// TIA Portal project "tamp" (V16)

(* hardware
DEVICE "S7-1200 station_1"  S7-1200 Station
   slot 0: "Rack_0"  S7-1200 Rack  Rack  V1.0
   slot 1: "PLC_1"  CPU 1212C AC/DC/Rly  6ES7 212-1BE40-0XB0  V4.0
*)

// ===== PLC "PLC_1"  CPU 1212C AC/DC/Rly =====

VAR_GLOBAL   // PLC tag table "Default tag table"
   "K1" AT %Q0.0 : Bool;
   "stop1" AT %I0.4 : Bool;
   "k2" AT %Q0.1 : Bool;
   "X" AT %M0.2 : Bool;
   "K3" AT %Q0.2 : Bool;
   "start1" AT %I0.2 : Bool;
   "Tag_2" AT %M0.1 : Bool;
   "start marker" AT %M0.3 : Bool;
   "stop marker" AT %M0.4 : Bool;
   "M 1 & 2" AT %M1.1 : Bool;
   "Tag_6" AT %M1.0 : Bool;
   "stop condition" AT %M0.5 : Bool;
   "STOP" AT %I0.3 : Bool;
   "L2" AT %I0.6 : Bool;
   "L3" AT %I0.7 : Bool;
   "L1" AT %I0.5 : Bool;
   "Tag_1" AT %MB20 : Byte;
   "Tag_3" AT %MB10 : USInt;
   "M 2 & 3" AT %M1.2 : Bool;
   "M 3 & 1" AT %M1.3 : Bool;
END_VAR

ORGANIZATION_BLOCK "Main"   // OB1, LAD, ProgramCycle
TITLE = "Main Program Sweep (Cycle)"
{ S7_Optimized_Access := 'TRUE' }
VERSION : 0.1
   VAR_INPUT
      Initial_Call : Bool;   // Initial call of this OB
      Remanence : Bool;   // =True, if remanent data are available
   END_VAR
   VAR_TEMP   // added for the SCL form of the ladder/FBD networks
      _w1 : Bool;
   END_VAR
BEGIN

REGION Network 1: start
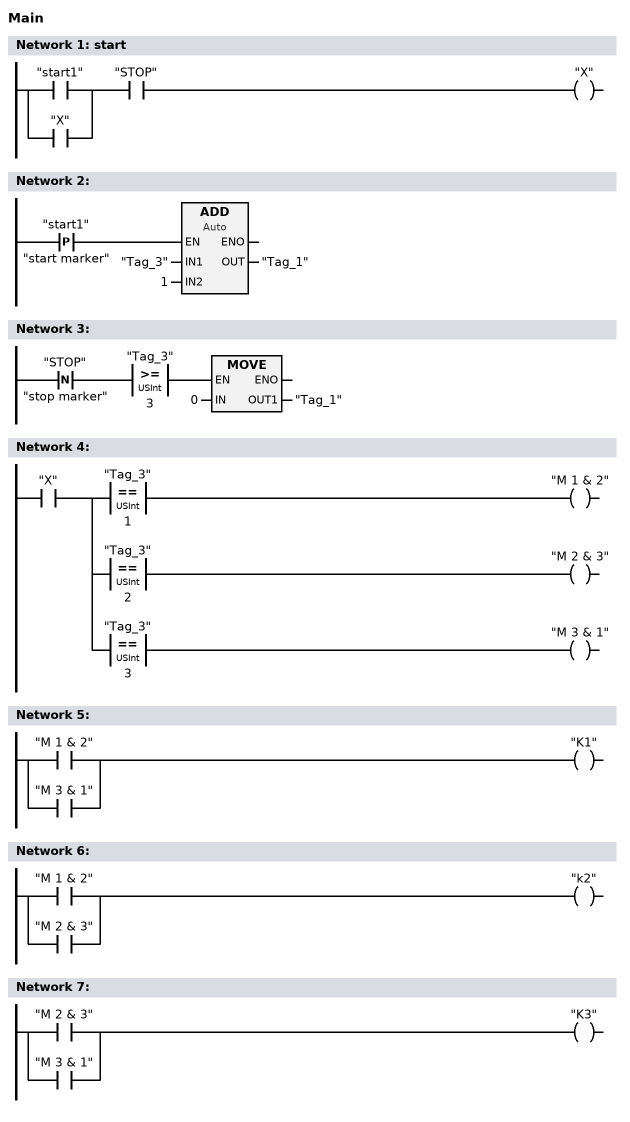
   RUNG wire#powerrail
      Contact( "start1" )
      wire#w1
      Contact( "STOP" )
      Coil( "X" )
   END_RUNG
   RUNG wire#powerrail
      Contact( "X" )
   END_RUNG wire#w1
   // the same network as SCL:
   "X" := ("start1" OR "X") AND "STOP";
END_REGION

REGION Network 2
   RUNG wire#powerrail
      P_Contact(operand := "start1", bit := "start marker")
      Add(in1 := "Tag_3", in2 := 1, out => "Tag_1")
   END_RUNG
   // the same network as SCL:
   #_w1 := "start1" AND NOT "start marker";   // rising edge of "start1"
   "start marker" := "start1";
   IF #_w1 THEN "Tag_1" := "Tag_3" + 1; END_IF;
END_REGION

REGION Network 3
   RUNG wire#powerrail
      N_Contact(operand := "STOP", bit := "stop marker")
      { S7_Templates := "SrcType := USInt" } GE_Contact(in1 := "Tag_3", in2 := 3)
      Move(in := 0, out1 => "Tag_1")
   END_RUNG
   // the same network as SCL:
   #_w1 := NOT "STOP" AND "stop marker";   // falling edge of "STOP"
   "stop marker" := "STOP";
   IF #_w1 AND ("Tag_3" >= 3) THEN "Tag_1" := 0; END_IF;
END_REGION

REGION Network 4
   RUNG wire#powerrail
      Contact( "X" )
      wire#w1
      { S7_Templates := "SrcType := USInt" } EQ_Contact(in1 := "Tag_3", in2 := 1)
      Coil( "M 1 & 2" )
   END_RUNG
   RUNG wire#w1
      { S7_Templates := "SrcType := USInt" } EQ_Contact(in1 := "Tag_3", in2 := 2)
      Coil( "M 2 & 3" )
   END_RUNG
   RUNG wire#w1
      { S7_Templates := "SrcType := USInt" } EQ_Contact(in1 := "Tag_3", in2 := 3)
      Coil( "M 3 & 1" )
   END_RUNG
   // the same network as SCL:
   "M 1 & 2" := "X" AND ("Tag_3" = 1);
   "M 2 & 3" := "X" AND ("Tag_3" = 2);
   "M 3 & 1" := "X" AND ("Tag_3" = 3);
END_REGION

REGION Network 5
   RUNG wire#powerrail
      Contact( "M 1 & 2" )
      wire#w1
      Coil( "K1" )
   END_RUNG
   RUNG wire#powerrail
      Contact( "M 3 & 1" )
   END_RUNG wire#w1
   // the same network as SCL:
   "K1" := "M 1 & 2" OR "M 3 & 1";
END_REGION

REGION Network 6
   RUNG wire#powerrail
      Contact( "M 1 & 2" )
      wire#w1
      Coil( "k2" )
   END_RUNG
   RUNG wire#powerrail
      Contact( "M 2 & 3" )
   END_RUNG wire#w1
   // the same network as SCL:
   "k2" := "M 1 & 2" OR "M 2 & 3";
END_REGION

REGION Network 7
   RUNG wire#powerrail
      Contact( "M 2 & 3" )
      wire#w1
      Coil( "K3" )
   END_RUNG
   RUNG wire#powerrail
      Contact( "M 3 & 1" )
   END_RUNG wire#w1
   // the same network as SCL:
   "K3" := "M 2 & 3" OR "M 3 & 1";
END_REGION
END_ORGANIZATION_BLOCK